FUNCTION F_GetStepperCommandMember : POINTER TO ST_StepperMotorCommand
VAR_INPUT
    nX : SINT;
    sY : STRING;
END_VAR
VAR
    i : INT;
    pResult: POINTER TO ST_StepperMotorCommand;
END_VAR

FOR i := 1 TO nEntryCount DO
    IF aLookupTable[i].nX = nX AND aLookupTable[i].sY = sY THEN
			pResult := aLookupTable[i].sCommand;
        EXIT;
    END_IF;
END_FOR;

F_GetStepperCommandMember := pResult;

END_FUNCTION

(* stored: Version 1.1.0.1, ProductVersion 3.1.4026.11
   POU F_GetStepperCommandMember: Id {9cd98949-e41e-4d8c-8a33-9e491ab78a2f}, SpecialFunc None *)
